// TIA Portal V19 export
DATA_BLOCK "DB_Schaltuhr"   // DB1050
{ S7_Optimized_Access := 'TRUE' }
// stored: AutoNumber false, MemoryReserve 0
   VAR RETAIN
      Tag : Array[1..7] of Struct   // Tag 1: Sonntag
         AZ_Begin1 : DTL;   // Arbeitszeit Beginn
         AZ_Ende1 : DTL;   // Arbeitszeit Ende
         AZ_Begin2 : DTL;   // Arbeitszeit Beginn
         AZ_Ende2 : DTL;   // Arbeitszeit Ende
      END_STRUCT;
      Tag_aktiv : Array[1..7] of Struct   // Übertagung aktiv- oder deaktivieren
         AZ_Begin1_aktiv : Bool;   // =1, das Wort wird im SPS übertragen (nach Plausibilitätsprüfung)
         AZ_Ende1_aktiv : Bool;   // =1, das Wort wird im SPS übertragen (nach Plausibilitätsprüfung)
         AZ_Begin2_aktiv : Bool;   // =1, das Wort wird im SPS übertragen (nach Plausibilitätsprüfung)
         AZ_Ende2_aktiv : Bool;   // =1, das Wort wird im SPS übertragen (nach Plausibilitätsprüfung)
      END_STRUCT;
      Date_Time_Visu : DTL;   // fürs Uhrzeit stellen
      BA_Visu : Int;
      SPS_Zeit_holen : Bool;
      SPS_Zeit_Stellen : Bool;
      Taste_uebernehmen : Bool;   // Schaltuhreinträge Prüfen und Übernehmen
      Uebernommen : Bool;   // für sichtbarkeit von Button "Übernehmen in Visu"
      nichtOK : Bool;   // Meldung generieren wenn Eintrag niO
   END_VAR
BEGIN
END_DATA_BLOCK
